# EPICS alarm handler configuration: mps_database/bare/alarms/areas/mpln_bsys_mp04.alhConfig
GROUP NULL MPLN:BSYS:MP04:1
$ALIAS MPS Link Node 202
$GUIDANCE
LTUH MPS
   Group Name: MPLN:BSYS:MP04:1
   Summary PV:  MPLN:BSYS:MP04:1:STATSUMY
$END
CHANNEL  MPLN:BSYS:MP04:1    MPLN:BSYS:MP04:1:MPS_EN_RBV		-----
CHANNEL  MPLN:BSYS:MP04:1    MPLN:BSYS:MP04:1:LC1_MODE_RBV		-----
GROUP NULL MPLN:BSYS:MP04:1
$ALIAS MPS Link Node 202
$GUIDANCE
LTUH MPS
   Group Name: MPLN:BSYS:MP04:1
   Summary PV:  MPLN:BSYS:MP04:1:STATSUMY
$END
CHANNEL  MPLN:BSYS:MP04:1    MPLN:BSYS:MP04:1:MPS_EN_RBV		-----
CHANNEL  MPLN:BSYS:MP04:1    MPLN:BSYS:MP04:1:LC1_MODE_RBV		-----
